Staubli VAL3: MainProg1.dtx

public dio dioIN = {link=fIn0}
public dio dioOUT = {link=fOut0}
public dio dioRotationON = {link=BasicIO-1\%Q0}
public dio dioRotationOFF = {link=BasicIO-1\%Q1}
public dio dioBuse = {link=BasicIO-1\%Q2}
public frame fPartCad = {x=0.000, y=0.000, z=0.000, rx=-0.000, ry=0.000, rz=-0.000, fatherId=world[0]}
public frame fCadToReal = {x=0, y=0, z=0, rx=0, ry=0, rz=0, fatherId=fPartCad[0]}
public mdesc mNomSpeed = {accel=100, vel=100, decel=100, tmax=99999, rmax=99999, blend=off, leave=50, reach=50}
public num nTraj
num nTimeStop
num nTimeStart
num nMode
num nEtat
public tool tCad = {x=0.000, y=0.000, z=0.000, rx=-0.000, ry=0.000, rz=-0.000, fatherId=flange[0], ioLink=valve1}
